(* Logix 5000 project; controller Injection_Comorfords vendor 1 type 14 code 222 rev 33.11; software revision 33.00 *)

TASK MainTask (continuous, watchdog 500 ms) : MainProgram
TASK SafetyTask (periodic, rate 20 ms, priority 10, watchdog 20 ms, safety) : SafetyProgram

MODULES
   Local : vendor 1 type 14 code 222 (5069 0, rev 33.11)
      WTU_C1_C2 : vendor 1 type 0 code 23 (Ethernet 192.168.2.12, rev 1.1)   // water tempering unit PLC
      WTU_C3_C4 : vendor 1 type 0 code 23 (Ethernet 192.168.2.13, rev 1.1)   // water tempering unit PLC
      PF525_Stirrer_Tank_1 : PowerFlex 525-EENET (Ethernet 192.168.2.15, rev 5.2, Output RPI 20 ms)   // 0.75 kW
      PF525_Feedingpump_1 : PowerFlex 525-EENET (Ethernet 192.168.2.16, rev 5.2, Output RPI 20 ms)   // 0.75 kW
      PF525_CIP_Pump_1 : PowerFlex 525-EENET (Ethernet 192.168.2.17, rev 5.2, Output RPI 20 ms)   // 0.75 kW
      PF525_Stirrer_Tank_2 : PowerFlex 525-EENET (Ethernet 192.168.2.18, rev 5.2, Output RPI 20 ms)   // 0.75 kW
      PF525_Feedingpump_2 : PowerFlex 525-EENET (Ethernet 192.168.2.19, rev 5.2, Output RPI 20 ms)   // 0.75 kW
      PF525_CIP_Pump_2 : PowerFlex 525-EENET (Ethernet 192.168.2.20, rev 5.2, Output RPI 20 ms)   // 0.75 kW
      Manifold_Cream : 2198-H008-ERS2 (Ethernet 192.168.2.22, rev 7.1, AMotionDiagnostics RPI 1 ms, CSafety_Output RPI 20 ms, DSafety_Input RPI 10 ms)
      Manifold_Jam : 2198-H008-ERS2 (Ethernet 192.168.2.23, rev 7.1, AMotionDiagnostics RPI 1 ms, CSafety_Output RPI 20 ms, DSafety_Input RPI 10 ms)
      X_Axis : 2198-H008-ERS2 (Ethernet 192.168.2.24, rev 7.1, AMotionDiagnostics RPI 1 ms, CSafety_Output RPI 20 ms, DSafety_Input RPI 10 ms)
      Z_Axis : 2198-H008-ERS2 (Ethernet 192.168.2.25, rev 7.1, AMotionDiagnostics RPI 1 ms, CSafety_Output RPI 20 ms, DSafety_Input RPI 10 ms)
      U2_MCC1_IO : 1734-AENTR (Ethernet 192.168.2.14, rev 6.1, Output RPI 20 ms)
         U2_MCC1_DIG_In_1 : 1734-IB8 (PointIO 3, rev 3.1)
         U2_MCC1_DIG_In_2 : 1734-IB8 (PointIO 4, rev 3.1)
         U2_MCC1_DIG_In_3 : 1734-IB8 (PointIO 5, rev 3.1)
         U2_MCC1_ANA_In_1 : vendor 1 type 115 code 210 (PointIO 6, rev 3.1, Input RPI 80 ms)
         U2_MCC1_DIG_Out_1 : vendor 1 type 7 code 231 (PointIO 7, rev 3.1)
         U2_MCC1_DIG_Out_2 : vendor 1 type 7 code 231 (PointIO 8, rev 3.1)
         U2_MCC1_DIG_Out_3 : 1734-OB8 (PointIO 9, rev 3.1)
         U2_MCC1_DIG_Out_4 : 1734-OB8 (PointIO 10, rev 3.1)
         U2_MCC1_DIG_Out_5 : 1734-OB8 (PointIO 11, rev 3.1)
         U2_MCC1_DIG_Out_6 : 1734-OB8 (PointIO 12, rev 3.1)
         U2_MCC1_Safety_DIG_In_1 : vendor 1 type 35 code 15 (PointIO 1, rev 2.1, Input RPI 10 ms, Output RPI 20 ms)
         U2_MCC1_Safety_DIG_Out_1 : vendor 1 type 35 code 16 (PointIO 2, rev 2.1, Input RPI 10 ms, Output RPI 20 ms)
      U5_MCC1_IO : 1734-AENTR (Ethernet 192.168.2.21, rev 6.1, Output RPI 20 ms)
         U5_MC1_DIG_In_1 : 1734-IB8 (PointIO 3, rev 3.1)
         U5_MC1_DIG_In_2 : 1734-IB8 (PointIO 4, rev 3.1)
         U5_MC1_DIG_In_3 : 1734-IB8 (PointIO 5, rev 3.1)
         U5_MC1_ANA_In_1 : 1734-IE4C (PointIO 6, rev 3.1, Input RPI 80 ms)
         U5_MC1_ANA_In_2 : 1734-IE4C (PointIO 7, rev 3.1, Input RPI 80 ms)
         U5_MC1_DIG_Out_1 : vendor 1 type 7 code 231 (PointIO 8, rev 3.1)
         U5_MC1_DIG_Out_2 : vendor 1 type 7 code 231 (PointIO 9, rev 3.1)
         U5_MC1_DIG_Out_3 : vendor 1 type 7 code 231 (PointIO 10, rev 3.1)
         U5_MC1_ANA_Out_1 : 1734-OE2C (PointIO 11, rev 3.1, Output RPI 80 ms)
         U5_MC1_Safety_DIG_Out_1 : vendor 1 type 35 code 16 (PointIO 2, rev 2.1, Output RPI 20 ms, Input RPI 10 ms)
         U5_MC1_Safety_DIG_In_1 : vendor 1 type 35 code 15 (PointIO 1, rev 2.1, Input RPI 10 ms, Output RPI 20 ms)
END_MODULES

VAR_GLOBAL   (* controller tags *)
   IA_2_1_LT01 : ALIAS FOR U2_MCC1_IO:6:I.Ch0Data;   // Level buffertank
   IA_2_1_PT01 : ALIAS FOR U2_MCC1_IO:6:I.Ch1Data;   // Pressure feeding pump 1
   IA_2_2_LT01 : ALIAS FOR U2_MCC1_IO:6:I.Ch2Data;   // Level buffertank
   IA_2_2_PT01 : ALIAS FOR U2_MCC1_IO:6:I.Ch3Data;   // Pressure feeding pump 1
   IA_5_1_PT01 : ALIAS FOR U5_MCC1_IO:6:I.Ch1Data;   // Pressure manifold Cream
   IA_5_1_PT02 : ALIAS FOR U5_MCC1_IO:6:I.Ch3Data;   // Pressure manifold Jam
   IA_5_1_TT01 : ALIAS FOR U5_MCC1_IO:6:I.Ch0Data;   // Temperature manifold Cream
   IA_5_1_TT02 : ALIAS FOR U5_MCC1_IO:6:I.Ch2Data;   // Temperature manifold Jam
   ID_2_1_GS01_1 : ALIAS FOR U2_MCC1_IO:4:I.1;   // Guard switch 1.1
   ID_2_1_GS01_2 : ALIAS FOR U2_MCC1_IO:4:I.2;   // Guard switch 1.2
   ID_2_1_GS01_3 : ALIAS FOR U2_MCC1_IO:4:I.3;   // Guard switch 1.3
   ID_2_1_LS01 : ALIAS FOR U2_MCC1_IO:4:I.5;   // Level switch feeding pump 1
   ID_2_1_OL_CIP : ALIAS FOR U2_MCC1_IO:4:I.6;   // Thermal overload CIP pump
   ID_2_1_OL_FAN : ALIAS FOR U2_MCC1_IO:3:I.0;   // Thermal overload Fan / Service socket
   ID_2_1_OL_M01 : ALIAS FOR U2_MCC1_IO:4:I.0;   // Thermal overload strirrer
   ID_2_1_OL_M02 : ALIAS FOR U2_MCC1_IO:4:I.4;   // Thermal overload feeding pump 1
   ID_2_1_PS01 : ALIAS FOR U2_MCC1_IO:3:I.1;   // Air pressure available
   ID_2_2_GS01_1 : ALIAS FOR U2_MCC1_IO:5:I.1;   // Guard switch 1.1
   ID_2_2_GS01_2 : ALIAS FOR U2_MCC1_IO:5:I.2;   // Guard switch 1.2
   ID_2_2_GS01_3 : ALIAS FOR U2_MCC1_IO:5:I.3;   // Guard switch 1.3
   ID_2_2_LS01 : ALIAS FOR U2_MCC1_IO:5:I.5;   // Level switch feeding pump 1
   ID_2_2_OL_CIP : ALIAS FOR U2_MCC1_IO:5:I.6;   // Thermal overload CIP pump
   ID_2_2_OL_M01 : ALIAS FOR U2_MCC1_IO:5:I.0;   // Thermal overload strirrer
   ID_2_2_OL_M02 : ALIAS FOR U2_MCC1_IO:5:I.4;   // Thermal overload feeding pump 1
   ID_4_1_GS03_1 : ALIAS FOR U5_MCC1_IO:5:I.0;   // Guard switch 3.1
   ID_4_1_GS03_2 : ALIAS FOR U5_MCC1_IO:5:I.1;   // Guard switch 3.2
   ID_4_1_GS03_3 : ALIAS FOR U5_MCC1_IO:5:I.2;   // Guard switch 3.3
   ID_4_1_GS04_1 : ALIAS FOR U5_MCC1_IO:5:I.3;   // Guard switch 4.1
   ID_4_1_GS04_2 : ALIAS FOR U5_MCC1_IO:5:I.4;   // Guard switch 4.2
   ID_4_1_GS04_3 : ALIAS FOR U5_MCC1_IO:5:I.5;   // Guard switch 4.3
   ID_5_1_GS01_1 : ALIAS FOR U5_MCC1_IO:4:I.0;   // Guard switch 1.1
   ID_5_1_GS01_2 : ALIAS FOR U5_MCC1_IO:4:I.1;   // Guard switch 1.2
   ID_5_1_GS01_3 : ALIAS FOR U5_MCC1_IO:4:I.2;   // Guard switch 1.3
   ID_5_1_GS02_1 : ALIAS FOR U5_MCC1_IO:4:I.3;   // Guard switch 2.1
   ID_5_1_GS02_2 : ALIAS FOR U5_MCC1_IO:4:I.4;   // Guard switch 2.2
   ID_5_1_GS02_3 : ALIAS FOR U5_MCC1_IO:4:I.5;   // Guard switch 2.3
   ID_5_1_OL_FAN : ALIAS FOR U5_MCC1_IO:3:I.0;   // Thermal overload Fan / Service socket
   ID_5_1_OL_M01 : ALIAS FOR U5_MCC1_IO:3:I.4;   // Thermal overload Power servo's
   ID_5_1_PS01 : ALIAS FOR U5_MCC1_IO:3:I.1;   // Air pressure available
   OA_5_1_CV01 : ALIAS FOR U5_MCC1_IO:11:O.Ch0Data;   // Pressure valve manifold Cream
   OA_5_1_CV02 : ALIAS FOR U5_MCC1_IO:11:O.Ch1Data;   // Pressure valve manifold Jam
   OD_2_1_CV01 : ALIAS FOR U2_MCC1_IO:9:O.0;   // Drain after tank
   OD_2_1_CV02 : ALIAS FOR U2_MCC1_IO:9:O.1;   // Bypass CIP before
   OD_2_1_CV03 : ALIAS FOR U2_MCC1_IO:9:O.2;   // Drain before CIP pump
   OD_2_1_CV04 : ALIAS FOR U2_MCC1_IO:9:O.3;   // Bypass CIP after
   OD_2_1_CV05 : ALIAS FOR U2_MCC1_IO:9:O.4;   // Before manifold
   OD_2_1_CV06 : ALIAS FOR U2_MCC1_IO:9:O.5;   // After manifold
   OD_2_1_CV07 : ALIAS FOR U2_MCC1_IO:9:O.6;   // Drain before tank
   OD_2_1_CV08 : ALIAS FOR U2_MCC1_IO:9:O.7;   // Sprinkler
   OD_2_1_CV09 : ALIAS FOR U2_MCC1_IO:10:O.0;   // Retour tank
   OD_2_1_CV10 : ALIAS FOR U2_MCC1_IO:10:O.1;   // Cold water inlet
   OD_2_1_CV11 : ALIAS FOR U2_MCC1_IO:10:O.2;   // Hot water inlet
   OD_2_1_CV12 : ALIAS FOR U2_MCC1_IO:10:O.3;   // Valve spare
   OD_2_1_CV13 : ALIAS FOR U2_MCC1_IO:10:O.4;   // Valve spare
   OD_2_1_CV14 : ALIAS FOR U2_MCC1_IO:10:O.5;   // Valve spare
   OD_2_1_CV15 : ALIAS FOR U2_MCC1_IO:10:O.6;   // Valve spare
   OD_2_1_CV16 : ALIAS FOR U2_MCC1_IO:10:O.7;   // Valve spare
   OD_2_1_GS01 : ALIAS FOR U2_MCC1_IO:8:O.0;   // Guard switch 1 lock
   OD_2_1_SLBZ : ALIAS FOR U2_MCC1_IO:7:O.3;   // Signal column BUZZER
   OD_2_1_SLGN : ALIAS FOR U2_MCC1_IO:7:O.0;   // Signal column GN
   OD_2_1_SLRD : ALIAS FOR U2_MCC1_IO:7:O.2;   // Signal column RD
   OD_2_1_SLYE : ALIAS FOR U2_MCC1_IO:7:O.1;   // Signal column YE
   OD_2_2_CV01 : ALIAS FOR U2_MCC1_IO:11:O.0;   // Drain after tank
   OD_2_2_CV02 : ALIAS FOR U2_MCC1_IO:11:O.1;   // Bypass CIP before
   OD_2_2_CV03 : ALIAS FOR U2_MCC1_IO:11:O.2;   // Drain before CIP pump
   OD_2_2_CV04 : ALIAS FOR U2_MCC1_IO:11:O.3;   // Bypass CIP after
   OD_2_2_CV05 : ALIAS FOR U2_MCC1_IO:11:O.4;   // Before manifold
   OD_2_2_CV06 : ALIAS FOR U2_MCC1_IO:11:O.5;   // After manifold
   OD_2_2_CV07 : ALIAS FOR U2_MCC1_IO:11:O.6;   // Drain before tank
   OD_2_2_CV08 : ALIAS FOR U2_MCC1_IO:11:O.7;   // Sprinkler
   OD_2_2_CV09 : ALIAS FOR U2_MCC1_IO:12:O.0;   // Retour tank
   OD_2_2_CV10 : ALIAS FOR U2_MCC1_IO:12:O.1;   // Cold water inlet
   OD_2_2_CV11 : ALIAS FOR U2_MCC1_IO:12:O.2;   // Hot water inlet
   OD_2_2_CV12 : ALIAS FOR U2_MCC1_IO:12:O.3;   // Valve spare
   OD_2_2_CV13 : ALIAS FOR U2_MCC1_IO:12:O.4;   // Valve spare
   OD_2_2_CV14 : ALIAS FOR U2_MCC1_IO:12:O.5;   // Valve spare
   OD_2_2_CV15 : ALIAS FOR U2_MCC1_IO:12:O.6;   // Valve spare
   OD_2_2_CV16 : ALIAS FOR U2_MCC1_IO:12:O.7;   // Valve spare
   OD_2_2_GS01 : ALIAS FOR U2_MCC1_IO:8:O.1;   // Guard switch 1 lock
   OD_4_1_GS01 : ALIAS FOR U5_MCC1_IO:9:O.0;   // Guard switch 1 lock
   OD_4_1_GS02 : ALIAS FOR U5_MCC1_IO:9:O.1;   // Guard switch 2 lock
   OD_4_1_GS03 : ALIAS FOR U5_MCC1_IO:9:O.2;   // Guard switch 3 lock
   OD_4_1_GS04 : ALIAS FOR U5_MCC1_IO:9:O.3;   // Guard switch 4 lock
   OD_5_1_CV01 : ALIAS FOR U5_MCC1_IO:10:O.0;   // Valve before manifold Cream
   OD_5_1_CV02 : ALIAS FOR U5_MCC1_IO:10:O.1;   // Valve before manifold Jam
   OD_5_1_SLBZ : ALIAS FOR U5_MCC1_IO:8:O.3;   // Signal column BUZZER
   OD_5_1_SLGN : ALIAS FOR U5_MCC1_IO:8:O.0;   // Signal column GN
   OD_5_1_SLRD : ALIAS FOR U5_MCC1_IO:8:O.2;   // Signal column RD
   OD_5_1_SLYE : ALIAS FOR U5_MCC1_IO:8:O.1;   // Signal column YE
END_VAR

PROGRAM MainProgram   (* main routine MainRoutine *)

ROUTINE MainRoutine   (* ladder *)
END_ROUTINE
END_PROGRAM

PROGRAM SafetyProgram   (* main routine MainRoutine, safety *)

ROUTINE MainRoutine   (* ladder *)
END_ROUTINE
END_PROGRAM
